FUNCTION_BLOCK FB_CondensingBoilerSystem
VAR_INPUT
END_VAR
VAR_OUTPUT
END_VAR
VAR
END_VAR

END_FUNCTION_BLOCK

(* stored: Version 1.1.0.1, ProductVersion 3.1.4024.10
   POU FB_CondensingBoilerSystem: Id {904c3c4f-e618-48ac-b2d2-67258d199066}, SpecialFunc None *)
